// TwinCAT 3 PLC project Untitled1
// ProgramVersion: 3.1.4023.0
// libraries:
//   Tc2_MC2, * (Beckhoff Automation GmbH)
//   Tc2_MC2_Drive, * (Beckhoff Automation GmbH)
//   Tc2_NC, * (Beckhoff Automation GmbH)
//   Tc2_Standard, * (Beckhoff Automation GmbH)
//   Tc2_System, * (Beckhoff Automation GmbH)
//   Tc3_Module, * (Beckhoff Automation GmbH)
// project tree:
//   GVLs/ link.TcGVL (not stored)
//   / PlcTask.TcTTO
//   POUs/ ControlParameters.TcPOU, ImpulseTest.TcPOU, leastSquare.TcPOU, MAIN.TcPOU, TorqueCounnter.TcPOU, torqueInput.TcPOU, velocityInput.TcPOU, velocityInput_.TcPOU, VelocityRide.TcPOU
// real-time tasks:
//   TASK PlcTask: cycle T#1ms, priority 8, ADS port 350
// motion (NC):
//   TASK NC-Task 1 SAF: cycle T#1ms, priority 4, ADS port 501
//   TASK NC-Task 1 SVB: cycle T#10ms, priority 10, ADS port 511
//   AXIS Axis 1 (id 1)
//     Dynamic: Acceleration=417.42, Deceleration=417.42, Jerk=1252.26
//     Velo: RefSearch=2.7828, RefSync=2.7828, SlowManual=13.914, FastManual=83.484, Fast=278.28, Maximum=278.28
//     OtherSettings: AllowMotionCmdToSlave=true
//     encoder EncType=19
//       EncPara: ScaleFactorNumerator=5, ScaleFactorDenominator=1048576, MaxCount=#xffffffff
//     drive DrvType=16
//       DrvPara: MaxCount=#xffffffff, DriveControlDWord=#x00020000
//         Analog: VeloReferenz=306.108, VeloScale=71.5255737304688, TorqueSetpointScale=10, ScaleFactorActTorque=0.1
//         TimeComp: TaskDelayCycles=1
//     controller CtrType=1
//       CtrPara: PriorControlFactor=1
//         PosDiffControl: Enable=false
//         Observer: BandWidth=20
//   AXIS Axis 2 (id 2)
//     Dynamic: Acceleration=417.42, Deceleration=417.42, Jerk=1252.26
//     Velo: RefSearch=2.7828, RefSync=2.7828, SlowManual=13.914, FastManual=83.484, Fast=278.28, Maximum=278.28
//     OtherSettings: AllowMotionCmdToSlave=true
//     encoder EncType=19
//       EncPara: ScaleFactorNumerator=5, ScaleFactorDenominator=1048576, MaxCount=#xffffffff
//     drive DrvType=16
//       DrvPara: MaxCount=#xffffffff, DriveControlDWord=#x00020000
//         Analog: VeloReferenz=306.108, VeloScale=71.5255737304688, TorqueSetpointScale=10, ScaleFactorActTorque=0.1
//         TimeComp: TaskDelayCycles=1
//     controller CtrType=1
//       CtrPara: PriorControlFactor=1
//         PosDiffControl: Enable=false
//         Observer: BandWidth=20
//   AXIS Axis 3 (id 3)
//     Dynamic: Acceleration=417.42, Deceleration=417.42, Jerk=1252.26
//     Velo: RefSearch=2.7828, RefSync=2.7828, SlowManual=13.914, FastManual=83.484, Fast=278.28, Maximum=278.28
//     OtherSettings: AllowMotionCmdToSlave=true
//     encoder EncType=19
//       EncPara: ScaleFactorNumerator=5, ScaleFactorDenominator=1048576, MaxCount=#xffffffff
//     drive DrvType=16
//       DrvPara: MaxCount=#xffffffff, DriveControlDWord=#x00000100
//         Analog: VeloReferenz=306.108, VeloScale=71.5255737304688, TorqueSetpointScale=10, ScaleFactorActTorque=0.1
//         TimeComp: TaskDelayCycles=1
//     controller CtrType=1
//       CtrPara: PriorControlFactor=1
//         Observer: BandWidth=20
//   AXIS Axis 4 (id 4)
//     OtherSettings: AllowMotionCmdToSlave=true
//     encoder EncType=19
//       EncPara: MaxCount=#xffffffff
//     drive DrvType=16
//       DrvPara: MaxCount=#xffffffff, DriveControlDWord=#x00000100
//         Analog: TorqueSetpointScale=10, ScaleFactorActTorque=0.1
//         TimeComp: TaskDelayCycles=1
//     controller CtrType=1
//       CtrPara: PriorControlFactor=1
//         Observer: BandWidth=20
// I/O:
//   DEVICE Device 5 (EtherCAT), AmsNetId 172.18.238.10.6.1
//     Term 1 (EK1100) [EK1100 EtherCAT Coupler (2A E-Bus)]
//       Term 2 (EL9221-5000) [EL9221-5000 Overcurrent protection 24V DC, 1Ch., max. 10A, adjustable]
//       Term 3 (EL1809) [EL1809 16Ch. Dig. Input 24V, 3ms]
//       Term 4 (EL2809) [EL2809 16Ch. Dig. Output 24V, 0.5A]
//       Term 5 (EL4028) [EL4028 8Ch. Ana. Output 4-20mA, 12bit]
//       Term 6 (EL3058) [EL3058 8Ch. Ana. Input 4-20mA]
//       Term 7 (EL3068) [EL3068 8Ch. Ana. Input 0-10V]
//       Term 8 (EL4008) [EL4008 8Ch. Ana. Output 0-10V, 12bit]
//       Term 9 (EL2634) [EL2634 4Ch. Relay Output, NO (250V AC / 30V DC)]
//       Term 10 (EL2634) [EL2634 4Ch. Relay Output, NO (250V AC / 30V DC)]
//       Term 11 (EL2634) [EL2634 4Ch. Relay Output, NO (250V AC / 30V DC)]
//       Term 15 (EL9011) [EL9011 End Terminal]
//     Term 12 (AX8640-0000-0103) [AX8640-0000-0103]
//       Drive 13 (AX8206-0000-0103) [AX8206-0000-0103]
//         modules: Device, Device, Device, Device, Device, Device, Device, Device, Device, Device, Device, Device, Device, Device, Device, Device, Device, Device, Device, Device, Device, Device, Device, Device, Device, Device, Device, Device, Device, Device, Device, Ch A, Ch A, Ch A, Ch A, Ch A, Ch A, Ch A, Ch A, Ch A, Ch A, Ch A, Ch A, Ch A, Ch A, Ch A, Ch A, Ch A, Ch A, Ch A, Ch A, Ch A, Ch A, Ch A, Ch A, Ch A, Ch A, Ch A, Ch B, Ch B, Ch B, Ch B, Ch B, Ch B, Ch B, Ch B, Ch B, Ch B, Ch B, Ch B, Ch B, Ch B, Ch B, Ch B, Ch B, Ch B, Ch B, Ch B, Ch B, Ch B, Ch B, Ch B, Ch B, Ch B, Ch B
//         startup 12992:1 := 414D383034312D78447830 // Ch A Motor parameters / Configured motor type
//         startup 24768:0 := FEFF // Ch A Interpolation sub mode select
//         startup 13000:5 := 0200 // Ch A Motor thermal model / Reaction
//         startup 12992:12 := 00803B45 // Ch A Motor parameters / Motor rated speed
//         startup 12992:13 := BC741340 // Ch A Motor parameters / Motor rated torque
//         startup 24694:0 := 48090000 // Ch A Motor standstill torque
//         startup 24800:0 := D007 // Ch A Positive torque/force limit value
//         startup 24801:0 := D007 // Ch A Negative torque/force limit value
//         startup 12288:6 := 4158383230362D303030302D30303030 // Ch A AxisMain parameters / Configured drive type
//         startup 12867:1 := 3333D33F // Ch A TorqueCtrl parameters / Configured channel rated current
//         startup 12867:2 := 66669E40 // Ch A TorqueCtrl parameters / Configured channel peak current
//         startup 12864:1 := C1059543 // Ch A TorqueCtrl parameters mappable / Torque control proportional gain q
//         startup 12864:2 := 8A0E7C39 // Ch A TorqueCtrl parameters mappable / Torque control integral action time q
//         startup 12608:1 := B246513D // Ch A VeloCtrl parameters mappable / Velocity control proportional gain
//         startup 12608:2 := 6F12033C // Ch A VeloCtrl parameters mappable / Velocity control integral action time
//         startup 12608:3 := 00980546 // Ch A VeloCtrl parameters mappable / Bipolar velocity limit value
//         startup 12992:15 := 0100 // Ch A Motor parameters / Motor temperature sensor connection
//         startup 12611:4 := 0100 // Ch A VeloCtrl observer / Observer type
//         startup 24672:0 := 08 // Ch A Modes of operation
//         startup 12296:2 := 00 // Ch A AxisMain parameters encoder polarity / Primary encoder actual values
//         startup 14016:1 := 414D383034312D78447830 // Ch B Motor parameters / Configured motor type
//         startup 26816:0 := FEFF // Ch B Interpolation sub mode select
//         startup 14024:5 := 0200 // Ch B Motor thermal model / Reaction
//         startup 14016:12 := 00803B45 // Ch B Motor parameters / Motor rated speed
//         startup 14016:13 := BC741340 // Ch B Motor parameters / Motor rated torque
//         startup 26742:0 := 48090000 // Ch B Motor standstill torque
//         startup 26848:0 := D007 // Ch B Positive torque/force limit value
//         startup 26849:0 := D007 // Ch B Negative torque/force limit value
//         startup 13312:6 := 4158383230362D303030302D30303030 // Ch B AxisMain parameters / Configured drive type
//         startup 13891:1 := 3333D33F // Ch B TorqueCtrl parameters / Configured channel rated current
//         startup 13891:2 := 66669E40 // Ch B TorqueCtrl parameters / Configured channel peak current
//         startup 13888:1 := C1059543 // Ch B TorqueCtrl parameters mappable / Torque control proportional gain q
//         startup 13888:2 := 8A0E7C39 // Ch B TorqueCtrl parameters mappable / Torque control integral action time q
//         startup 13632:1 := B246513D // Ch B VeloCtrl parameters mappable / Velocity control proportional gain
//         startup 13632:2 := 6F12033C // Ch B VeloCtrl parameters mappable / Velocity control integral action time
//         startup 13632:3 := 00980546 // Ch B VeloCtrl parameters mappable / Bipolar velocity limit value
//         startup 14016:15 := 0100 // Ch B Motor parameters / Motor temperature sensor connection
//         startup 13635:4 := 0100 // Ch B VeloCtrl observer / Observer type
//         startup 26720:0 := 08 // Ch B Modes of operation
//         startup 13320:2 := 00 // Ch B AxisMain parameters encoder polarity / Primary encoder actual values
//       Drive 14 (AX8206-0000-0103) [AX8206-0000-0103]
//         modules: Device, Device, Device, Device, Device, Device, Device, Device, Device, Device, Device, Device, Device, Device, Device, Device, Device, Device, Device, Device, Device, Device, Device, Device, Device, Device, Device, Device, Device, Device, Device, Ch A, Ch A, Ch A, Ch A, Ch A, Ch A, Ch A, Ch A, Ch A, Ch A, Ch A, Ch A, Ch A, Ch A, Ch A, Ch A, Ch A, Ch A, Ch A, Ch A, Ch A, Ch A, Ch A, Ch A, Ch A, Ch A, Ch A, Ch B, Ch B, Ch B, Ch B, Ch B, Ch B, Ch B, Ch B, Ch B, Ch B, Ch B, Ch B, Ch B, Ch B, Ch B, Ch B, Ch B, Ch B, Ch B, Ch B, Ch B, Ch B, Ch B, Ch B, Ch B, Ch B
//         startup 12992:1 := 414D383034312D78447831 // Ch A Motor parameters / Configured motor type
//         startup 24768:0 := FEFF // Ch A Interpolation sub mode select
//         startup 13000:5 := 0200 // Ch A Motor thermal model / Reaction
//         startup 12992:12 := 00803B45 // Ch A Motor parameters / Motor rated speed
//         startup 12992:13 := BC741340 // Ch A Motor parameters / Motor rated torque
//         startup 24694:0 := 48090000 // Ch A Motor standstill torque
//         startup 24800:0 := D007 // Ch A Positive torque/force limit value
//         startup 24801:0 := D007 // Ch A Negative torque/force limit value
//         startup 12288:6 := 4158383230362D303030302D30303030 // Ch A AxisMain parameters / Configured drive type
//         startup 12867:1 := 3333D33F // Ch A TorqueCtrl parameters / Configured channel rated current
//         startup 12867:2 := 66669E40 // Ch A TorqueCtrl parameters / Configured channel peak current
//         startup 12864:1 := C1059543 // Ch A TorqueCtrl parameters mappable / Torque control proportional gain q
//         startup 12864:2 := 8A0E7C39 // Ch A TorqueCtrl parameters mappable / Torque control integral action time q
//         startup 12608:1 := 7409A73D // Ch A VeloCtrl parameters mappable / Velocity control proportional gain
//         startup 12608:2 := 6F12033C // Ch A VeloCtrl parameters mappable / Velocity control integral action time
//         startup 12608:3 := 00980546 // Ch A VeloCtrl parameters mappable / Bipolar velocity limit value
//         startup 12992:15 := 0100 // Ch A Motor parameters / Motor temperature sensor connection
//         startup 12611:4 := 0100 // Ch A VeloCtrl observer / Observer type
//         startup 24672:0 := 08 // Ch A Modes of operation
//         startup 12296:2 := 00 // Ch A AxisMain parameters encoder polarity / Primary encoder actual values
//       Term 16 (EL9011) [EL9011 End Terminal]
// variable links:
//   Device 5 (EtherCAT) <-> Device 5 (EtherCAT)/Term 12 (AX8640-0000-0103)/Drive 13 (AX8206-0000-0103)
//     Term 12 (AX8640-0000-0103)/PSM Controlword for axis/Controlword for axis <-> Device/DeviceMain Outputs/Power supply controlword
//   Device 5 (EtherCAT) <-> Device 5 (EtherCAT)/Term 12 (AX8640-0000-0103)/Drive 14 (AX8206-0000-0103)
//     Term 12 (AX8640-0000-0103)/PSM Controlword for axis/Controlword for axis <-> Device/DeviceMain Outputs/Power supply controlword
//   NC-Task 1 SAF/Axes/Axis 1 <-> Device 5 (EtherCAT)/Term 12 (AX8640-0000-0103)/Drive 13 (AX8206-0000-0103)
//     Drive/Inputs/In/nDataIn1 <-> Ch A/Ch A PositionControl Inputs/Ch A Following error actual value
//     Drive/Inputs/In/nDataIn3[0] <-> Ch A/Ch A TorqueControl Inputs/Ch A Torque/force actual value
//     Drive/Inputs/In/nDcOutputTime <-> InfoData/DcOutputShift
//     Drive/Inputs/In/nState1 <-> Ch A/Ch A AxisMain Inputs/Ch A Statusword
//     Drive/Inputs/In/nState2 <-> Ch A/Ch A AxisMain Inputs/Ch A Statusword @bit 8
//     Drive/Inputs/In/nState4 @bit 1 <-> WcState/InputToggle
//     Drive/Inputs/In/nState4 <-> WcState/WcState
//     Drive/Outputs/Out/nCtrl1 <-> Ch A/Ch A AxisMain Outputs/Ch A Controlword
//     Drive/Outputs/Out/nCtrl2 <-> Ch A/Ch A AxisMain Outputs/Ch A Controlword @bit 8
//     Drive/Outputs/Out/nDataOut1 <-> Ch A/Ch A Interpolator Outputs/Ch A Target position
//     Enc/Inputs/In/nDataIn1 <-> Ch A/Ch A AxisMain Inputs/Ch A Position actual value
//     Enc/Inputs/In/nDataIn7 <-> Ch A/Ch A AxisMain Inputs/Ch A Velocity actual value
//     Enc/Inputs/In/nDcInputTime <-> InfoData/DcInputShift
//     Enc/Inputs/In/nState2 @bit 5 <-> Ch A/Ch A AxisMain Inputs/Position actual value invalid
//     Enc/Inputs/In/nState4 @bit 1 <-> WcState/InputToggle
//     Enc/Inputs/In/nState4 <-> WcState/WcState
//   NC-Task 1 SAF/Axes/Axis 2 <-> Device 5 (EtherCAT)/Term 12 (AX8640-0000-0103)/Drive 13 (AX8206-0000-0103)
//     Drive/Inputs/In/nDataIn1 <-> Ch B/Ch B PositionControl Inputs/Ch B Following error actual value
//     Drive/Inputs/In/nDataIn3[0] <-> Ch B/Ch B TorqueControl Inputs/Ch B Torque/force actual value
//     Drive/Inputs/In/nDcOutputTime <-> InfoData/DcOutputShift
//     Drive/Inputs/In/nState1 <-> Ch B/Ch B AxisMain Inputs/Ch B Statusword
//     Drive/Inputs/In/nState2 <-> Ch B/Ch B AxisMain Inputs/Ch B Statusword @bit 8
//     Drive/Inputs/In/nState4 @bit 1 <-> WcState/InputToggle
//     Drive/Inputs/In/nState4 <-> WcState/WcState
//     Drive/Outputs/Out/nCtrl1 <-> Ch B/Ch B AxisMain Outputs/Ch B Controlword
//     Drive/Outputs/Out/nCtrl2 <-> Ch B/Ch B AxisMain Outputs/Ch B Controlword @bit 8
//     Drive/Outputs/Out/nDataOut1 <-> Ch B/Ch B Interpolator Outputs/Ch B Target position
//     Enc/Inputs/In/nDataIn1 <-> Ch B/Ch B AxisMain Inputs/Ch B Position actual value
//     Enc/Inputs/In/nDataIn7 <-> Ch B/Ch B AxisMain Inputs/Ch B Velocity actual value
//     Enc/Inputs/In/nDcInputTime <-> InfoData/DcInputShift
//     Enc/Inputs/In/nState2 @bit 5 <-> Ch B/Ch B AxisMain Inputs/Position actual value invalid
//     Enc/Inputs/In/nState4 @bit 1 <-> WcState/InputToggle
//     Enc/Inputs/In/nState4 <-> WcState/WcState
//   NC-Task 1 SAF/Axes/Axis 3 <-> Device 5 (EtherCAT)/Term 12 (AX8640-0000-0103)/Drive 14 (AX8206-0000-0103)
//     Drive/Inputs/In/nDataIn1 <-> Ch A/Ch A PositionControl Inputs/Ch A Following error actual value
//     Drive/Inputs/In/nDataIn3[0] <-> Ch A/Ch A TorqueControl Inputs/Ch A Torque/force actual value
//     Drive/Inputs/In/nDcOutputTime <-> InfoData/DcOutputShift
//     Drive/Inputs/In/nState1 <-> Ch A/Ch A AxisMain Inputs/Ch A Statusword
//     Drive/Inputs/In/nState2 <-> Ch A/Ch A AxisMain Inputs/Ch A Statusword @bit 8
//     Drive/Inputs/In/nState4 @bit 1 <-> WcState/InputToggle
//     Drive/Inputs/In/nState4 <-> WcState/WcState
//     Drive/Outputs/Out/nCtrl1 <-> Ch A/Ch A AxisMain Outputs/Ch A Controlword
//     Drive/Outputs/Out/nCtrl2 <-> Ch A/Ch A AxisMain Outputs/Ch A Controlword @bit 8
//     Enc/Inputs/In/nDataIn1 <-> Ch A/Ch A AxisMain Inputs/Ch A Position actual value
//     Enc/Inputs/In/nDataIn7 <-> Ch A/Ch A AxisMain Inputs/Ch A Velocity actual value
//     Enc/Inputs/In/nDcInputTime <-> InfoData/DcInputShift
//     Enc/Inputs/In/nState2 @bit 5 <-> Ch A/Ch A AxisMain Inputs/Position actual value invalid
//     Enc/Inputs/In/nState4 @bit 1 <-> WcState/InputToggle
//     Enc/Inputs/In/nState4 <-> WcState/WcState
//   NC-Task 1 SAF/Axes/Axis 4 <-> Device 5 (EtherCAT)/Term 12 (AX8640-0000-0103)/Drive 14 (AX8206-0000-0103)
//     Drive/Inputs/In/nDataIn1 <-> Ch B/Ch B PositionControl Inputs/Ch B Following error actual value
//     Drive/Inputs/In/nState1 <-> Ch B/Ch B AxisMain Inputs/Ch B Statusword
//     Drive/Inputs/In/nState2 <-> Ch B/Ch B AxisMain Inputs/Ch B Statusword @bit 8
//     Drive/Outputs/Out/nCtrl1 <-> Ch B/Ch B AxisMain Outputs/Ch B Controlword
//     Drive/Outputs/Out/nCtrl2 <-> Ch B/Ch B AxisMain Outputs/Ch B Controlword @bit 8
//     Enc/Inputs/In/nDataIn1 <-> Ch B/Ch B AxisMain Inputs/Ch B Position actual value
//     Enc/Inputs/In/nState2 @bit 5 <-> Ch B/Ch B AxisMain Inputs/Position actual value invalid
//   Untitled1/Untitled1 Instance <-> Device 5 (EtherCAT)/Term 12 (AX8640-0000-0103)/Drive 13 (AX8206-0000-0103)
//     PlcTask Outputs/link.torqueOfsetX <-> Ch A/Ch A TorqueControl Outputs/Ch A Torque/force offset
//     PlcTask Outputs/link.torqueOfsetY <-> Ch B/Ch B TorqueControl Outputs/Ch B Torque/force offset
//     PlcTask Outputs/link.torqueX <-> Ch A/Ch A TorqueControl Outputs/Ch A Target torque/force
//     PlcTask Outputs/link.torqueY <-> Ch B/Ch B TorqueControl Outputs/Ch B Target torque/force
//     PlcTask Outputs/link.xAxisVelocity <-> Ch A/Ch A Interpolator Outputs/Ch A Target velocity
//     PlcTask Outputs/link.yAxisVelocity <-> Ch B/Ch B Interpolator Outputs/Ch B Target velocity
//   Untitled1/Untitled1 Instance <-> Device 5 (EtherCAT)/Term 12 (AX8640-0000-0103)/Drive 14 (AX8206-0000-0103)
//     PlcTask Outputs/link.zAxisVelocity <-> Ch A/Ch A Interpolator Outputs/Ch A Target velocity
//   Untitled1/Untitled1 Instance <-> NC-Task 1 SAF/Axes/Axis 1
//     PlcTask Inputs/MAIN.setAxis[0].NcToPlc <-> Outputs/ToPlc
//     PlcTask Outputs/MAIN.setAxis[0].PlcToNc <-> Inputs/FromPlc
//   Untitled1/Untitled1 Instance <-> NC-Task 1 SAF/Axes/Axis 2
//     PlcTask Inputs/MAIN.setAxis[1].NcToPlc <-> Outputs/ToPlc
//     PlcTask Outputs/MAIN.setAxis[1].PlcToNc <-> Inputs/FromPlc
//   Untitled1/Untitled1 Instance <-> NC-Task 1 SAF/Axes/Axis 3
//     PlcTask Inputs/MAIN.setAxis[2].NcToPlc <-> Outputs/ToPlc
//     PlcTask Outputs/MAIN.setAxis[2].PlcToNc <-> Inputs/FromPlc

CONFIGURATION Untitled1
    RESOURCE PLC ON TwinCAT3
        TASK PlcTask(INTERVAL := T#500us, PRIORITY := 8);
        PROGRAM MAIN WITH PlcTask : MAIN;
        PROGRAM leastSquare WITH PlcTask : leastSquare;
        PROGRAM velocityInput_ WITH PlcTask : velocityInput_;
        PROGRAM velocityInput WITH PlcTask : velocityInput;
        PROGRAM torqueInput WITH PlcTask : torqueInput;
        PROGRAM ImpulseTest WITH PlcTask : ImpulseTest;
        PROGRAM VelocityRide WITH PlcTask : VelocityRide;
    END_RESOURCE
END_CONFIGURATION

// ---- POUs/MAIN.TcPOU
PROGRAM MAIN
VAR
	sampleTime: REAL := 0.5;
	state: INT	:=	0;	
	start: BOOL	:=	FALSE;
	operationModeWrite: SINT	:=	10;	
	
	{attribute 'TcNcAxis' := '[0]:=Axis 1;[1]:=Axis 2;[2]:=Axis 3'} 
    // Using an axis in an array.
    setAxis     : ARRAY [0..2] OF AXIS_REF;
	
	opertionModeRead: SINT;
	
	fbCoERead: FB_CoERead;
	
	MotorEnable: BOOL:=FALSE;
	
	mcReset: MC_Reset;
	mcPower: MC_Power;
	
////////
	
	operitonModeCh: WORD;
	subIndex: BYTE;	
	axisSelect: (xAxis, yAxis, zAxis, xyAxis, allAxis);	
	fbCoEWrite: FB_CoEWrite;	
	//torque : FB_TorqueInput;
	
END_VAR
VAR_INPUT
	dummy : INT ;
END_VAR

CASE state OF
	//Axis Selection
0:
	IF start THEN
		
		IF axisSelect = xAxis THEN
			operitonModeCh := 16#6060;
			subIndex := 0;
			MotorEnable:=TRUE;
			dummy := 0;	
		ELSIF axisSelect = yAxis THEN	
			operitonModeCh := 16#6860;		
			subIndex := 0;
			MotorEnable:=TRUE;	
			dummy := 1;	
		ELSIF axisSelect = zAxis THEN	
			operitonModeCh := 16#6860;
			MotorEnable:=TRUE;	
			dummy := 2;
			subIndex := 0;
			
		ELSIF axisSelect = xyAxis THEN	
			operitonModeCh := 16#6860;
			MotorEnable:=TRUE;	
			dummy := 3;
			subIndex := 0;
		END_IF
		
		state:=190;
		start:=FALSE;		
	END_IF

190:
	mcReset(
	Axis:=setAxis[dummy] , 
	Execute:=TRUE , 
	 );
	IF NOT mcReset.Busy AND mcReset.Done THEN		
		mcReset(Axis:=setAxis[dummy], Execute:=FALSE);		
		state:=200;
	END_IF
	
	//Mod of operation
200:


	fbCoEWrite(
		Axis:= setAxis[dummy], 
		NetId:='', 
		Index:= operitonModeCh, 
		SubIndex:=subIndex,
		pSrcBuf:= ADR(operationModeWrite), 
		BufLen:= SIZEOF(operationModeWrite), 
		Execute:=TRUE , 		
		CompleteAccess:=TRUE , 
		 );
		
	IF NOT fbCoEWrite.Busy THEN
		fbCoEWrite(
		Axis:= setAxis[dummy], 
		NetId:='', 
		Index:= operitonModeCh, 
		SubIndex:=subIndex, 
		pSrcBuf:= ADR(operationModeWrite), 
		BufLen:= SIZEOF(operationModeWrite), 
		Execute:=FALSE , 		
		CompleteAccess:=TRUE , 
		 );
		
		fbCoERead(
			Axis:=setAxis[dummy] , 
			NetId:= '', 
			Index:= operitonModeCh,
			SubIndex:= subIndex,
			pDstBuf:= ADR(opertionModeRead), 
			BufLen:= SIZEOF(opertionModeRead), 
			Execute:= TRUE, 			
			CompleteAccess:=TRUE , 
			 );
			
			IF opertionModeRead = operationModeWrite AND NOT fbCoERead.Busy THEN
			
				fbCoeRead(Axis:=setAxis[dummy],Execute:=FALSE );
				IF NOT fbCoERead.Execute THEN
					state:=210;
				END_IF
			END_IF
	END_IF
	
	//power enable
	//motor enable
210:
	mcReset(
	Axis:=setAxis[dummy] , 
	Execute:=TRUE , 
	 );
	IF NOT mcReset.Busy AND mcReset.Done THEN		
		mcReset(Axis:=setAxis[dummy], Execute:=FALSE);		
		state:=220;
	END_IF
	
	220:
	
	mcPower(
	Axis:=setAxis[dummy] , 
	Enable:= MotorEnable , 
	Enable_Positive:= MotorEnable, 
	Enable_Negative:= MotorEnable, 
 );
	IF (mcPower.Status AND MotorEnable) OR (NOT mcPower.Status AND NOT MotorEnable) THEN 

		state:=230;
	END_IF
	

230:

// 	torque(torqueInput:=20, duration:=2);
//	IF torque.busy = FALSE THEN
//		state := 232;
//	END_IF

 
232:
  
// velocityInput();
// IF NOT velocityInput.busy THEN
//	 state := 240;
// END_IF
 
240 :
 mcReset(
	Axis:=setAxis[dummy] , 
	Execute:=TRUE , 
	 );
	IF NOT mcReset.Busy AND mcReset.Done THEN		
		mcReset(Axis:=setAxis[dummy], Execute:=FALSE);		
		state:=250;
	END_IF
 
	250:
 	MotorEnable := FALSE;
 	mcPower(
	Axis:=setAxis[dummy] , 
	Enable:= MotorEnable , 
	Enable_Positive:= MotorEnable, 
	Enable_Negative:= MotorEnable, 
 );
	IF (mcPower.Status AND MotorEnable) OR (NOT mcPower.Status AND NOT MotorEnable) THEN 
		state:=260;
	END_IF
	//Motor disable
260:
 	

	state := 0;

END_CASE

END_PROGRAM

// ---- POUs/leastSquare.TcPOU
PROGRAM leastSquare
VAR
	state: USINT := 0;
	Torque_Nm :REAL := 0.5;
	duration :INT :=10000;
	startTest :BOOL := FALSE;	
	TorquePerThousand: INT;		

	TorqueCounter: INT;
	TorqInterval: INT;
END_VAR

CASE state OF
	
0 :
	
	IF MAIN.dummy = 0 AND startTest  THEN
		state := 10;
	ELSIF MAIN.dummy = 1 AND startTest THEN
		state := 30;
	END_IF	

	10: //varying amplitude squarewaves for least square
			IF startTest THEN
				TorqueCounter := TorqueCounter + 1;
				IF TorqueCounter < TorqInterval THEN
					link.torqueX := TO_INT(Torque_Nm * 1/2.37*1000);
				ELSIF TorqueCounter >= TorqInterval AND TorqueCounter <TorqInterval*2 THEN
					link.torqueX := TO_INT(-Torque_Nm *1/2.37*1000);
				ELSIF TorqueCounter >= TorqInterval*2 AND TorqueCounter <TorqInterval*3 THEN
					link.torqueX := TO_INT(Torque_Nm * 2/2.37*1000); 
				ELSIF TorqueCounter >= TorqInterval*3 AND TorqueCounter <TorqInterval*4 THEN
					link.torqueX := TO_INT(-Torque_Nm * 2/2.37*1000);
				ELSIF TorqueCounter >= TorqInterval*4 AND TorqueCounter <TorqInterval*5 THEN
					link.torqueX := TO_INT(Torque_Nm * 3/2.37*1000); 
				ELSIF TorqueCounter >= TorqInterval*5 AND TorqueCounter <TorqInterval*6 THEN
					link.torqueX := TO_INT(-Torque_Nm * 3/2.37*1000);
				ELSIF TorqueCounter >= TorqInterval*6 AND TorqueCounter <TorqInterval*7 THEN
					link.torqueX := TO_INT(Torque_Nm * 4/2.37*1000); 
					
				ELSIF TorqueCounter >= TorqInterval*7 AND TorqueCounter <TorqInterval*8 THEN
					link.torqueX := TO_INT(-Torque_Nm * 4/2.37*1000);		
				ELSIF TorqueCounter >= TorqInterval*8 AND TorqueCounter <TorqInterval*9 THEN
					link.torqueX := TO_INT(Torque_Nm * 3/2.37*1000); 
				ELSIF TorqueCounter >= TorqInterval*9 AND TorqueCounter <TorqInterval*10 THEN
					link.torqueX := TO_INT(-Torque_Nm * 3/2.37*1000);
				ELSIF TorqueCounter >= TorqInterval*10 AND TorqueCounter <TorqInterval*11 THEN
					link.torqueX := TO_INT(Torque_Nm * 2/2.37*1000); 
				ELSIF TorqueCounter >= TorqInterval*11 AND TorqueCounter <TorqInterval*12 THEN
					link.torqueX := TO_INT(-Torque_Nm * 2/2.37*1000);
				ELSIF TorqueCounter >= TorqInterval*12 AND TorqueCounter <TorqInterval*13 THEN
					link.torqueX := TO_INT(Torque_Nm * 1/2.37*1000); 
				ELSIF TorqueCounter >= TorqInterval*13 AND TorqueCounter <TorqInterval*14 THEN
					link.torqueX := TO_INT(-Torque_Nm * 1/2.37*1000);
				ELSIF TorqueCounter >= TorqInterval*14 THEN
					link.torqueX := 0;
					state:=60;
				END_IF
		ELSE
		link.torqueX := 0;		
		startTest := FALSE;
		TorqueCounter := 0;
		state := 60;
		
		END_IF
	30: //varying amplitude squarewaves for least square
			IF startTest THEN
				TorqueCounter := TorqueCounter + 1;
				IF TorqueCounter < TorqInterval THEN
					link.torqueY := TO_INT(Torque_Nm * 0.5/2.37*1000);
				ELSIF TorqueCounter >= TorqInterval AND TorqueCounter <TorqInterval*2 THEN
					link.torqueY := TO_INT(-Torque_Nm *0.5/2.37*1000);
				ELSIF TorqueCounter >= TorqInterval*2 AND TorqueCounter <TorqInterval*3 THEN
					link.torqueY := TO_INT(Torque_Nm * 1/2.37*1000); 
				ELSIF TorqueCounter >= TorqInterval*3 AND TorqueCounter <TorqInterval*4 THEN
					link.torqueY := TO_INT(-Torque_Nm * 1/2.37*1000);
				ELSIF TorqueCounter >= TorqInterval*4 AND TorqueCounter <TorqInterval*5 THEN
					link.torqueY := TO_INT(Torque_Nm * 1.5/2.37*1000); 
				ELSIF TorqueCounter >= TorqInterval*5 AND TorqueCounter <TorqInterval*6 THEN
					link.torqueY := TO_INT(-Torque_Nm * 1.5/2.37*1000);
				ELSIF TorqueCounter >= TorqInterval*6 AND TorqueCounter <TorqInterval*7 THEN
					link.torqueY := TO_INT(Torque_Nm * 2/2.37*1000); 
				ELSIF TorqueCounter >= TorqInterval*7 AND TorqueCounter <TorqInterval*8 THEN
					link.torqueY := TO_INT(-Torque_Nm * 2/2.37*1000); 	
				ELSIF TorqueCounter >= TorqInterval*8 AND TorqueCounter <TorqInterval*9 THEN
					link.torqueY := TO_INT(Torque_Nm * 2.5/2.37*1000); 				
				ELSIF TorqueCounter >= TorqInterval*9 AND TorqueCounter <TorqInterval*10 THEN
					link.torqueY := TO_INT(-Torque_Nm * 2.5/2.37*1000); 					

				ELSIF TorqueCounter >= TorqInterval*10 AND TorqueCounter <TorqInterval*11 THEN
					link.torqueY := TO_INT(Torque_Nm * 2/2.37*1000); 					
				ELSIF TorqueCounter >= TorqInterval*11 AND TorqueCounter <TorqInterval*12 THEN
					link.torqueY := TO_INT(-Torque_Nm * 2/2.37*1000);							
				ELSIF TorqueCounter >= TorqInterval*12 AND TorqueCounter <TorqInterval*13 THEN
					link.torqueY := TO_INT(Torque_Nm * 1.5/2.37*1000);			
				ELSIF TorqueCounter >= TorqInterval*13 AND TorqueCounter <TorqInterval*14 THEN
					link.torqueY := TO_INT(-Torque_Nm * 1.5/2.37*1000);		
				ELSIF TorqueCounter >= TorqInterval*14 AND TorqueCounter <TorqInterval*15 THEN
					link.torqueY := TO_INT(Torque_Nm * 1/2.37*1000); 
				ELSIF TorqueCounter >= TorqInterval*15 AND TorqueCounter <TorqInterval*16 THEN
					link.torqueY := TO_INT(-Torque_Nm * 1/2.37*1000);
				ELSIF TorqueCounter >= TorqInterval*16 AND TorqueCounter <TorqInterval*17 THEN
					link.torqueY := TO_INT(Torque_Nm * 0.5/2.37*1000); 
				ELSIF TorqueCounter >= TorqInterval*17 AND TorqueCounter <TorqInterval*18 THEN
					link.torqueY := TO_INT(-Torque_Nm * 0.5/2.37*1000);
				ELSIF TorqueCounter >= TorqInterval*18 THEN
					link.torqueY := 0;
					state:=60;
				END_IF
		ELSE
		link.torqueY := 0;		
		startTest := FALSE;
		TorqueCounter := 0;
		state := 60;
		
		END_IF
	
	
60 :
	startTest:= FALSE;
	state :=0;
	TorqueCounter := 0;
END_CASE

END_PROGRAM

// ---- POUs/velocityInput_.TcPOU
PROGRAM velocityInput_
VAR
	
	velocityStarter : BOOL := FALSE;
	state : INT := 0;	
	counter : LREAL := 0;
	bias : LREAL :=0.4;
	duration: REAL := 30000;
	velocityInput: INT:= -1;
	f0 :LREAL	:=0;
	f1 :LREAL:=100;
	T : LREAL ;	
	x: LREAL;	
	


END_VAR

CASE state OF

0 :
	
	IF MAIN.dummy = 0 AND velocityStarter  THEN
		state := 10;
	ELSIF MAIN.dummy = 1 AND velocityStarter THEN
		state := 30;
	END_IF	
		
10 : 

	IF velocityStarter THEN		
		
		IF counter < duration THEN
			T :=duration/1000.0;
			x:=SIN(2*pi*((f0*counter/1000)+((f1-f0)/(2*T)*(EXPT(counter/1000,2)))));
			link.xAxisVelocity := LREAL_TO_DINT((velocityInput*10000/(5)*60)*(x+bias/(velocityInput)));
		ELSE
			link.xAxisVelocity := 0;
			state := 60;
		END_IF
		counter := counter + MAIN.sampleTime;
	ELSE
		link.xAxisVelocity := 0;
	
	END_IF
	
30:
	IF velocityStarter THEN		
		
		IF counter < duration THEN
			T :=duration/1000.0;
			x:=SIN(2*pi*((f0*counter/1000)+((f1-f0)/(2*T)*(EXPT(counter/1000,2)))));
			link.yAxisVelocity := LREAL_TO_DINT((velocityInput*10000/(5)*60)*(x+bias/(velocityInput)));
		ELSE
			link.yAxisVelocity := 0;
			state := 60;
		END_IF
		counter := counter + MAIN.sampleTime;
	ELSE
		link.yAxisVelocity := 0;
	
	END_IF

60 :
	velocityStarter:= FALSE;
	state :=0;
	counter := 0;
END_CASE

END_PROGRAM

// ---- POUs/velocityInput.TcPOU
PROGRAM velocityInput
VAR
	velocityStarter : BOOL := FALSE;
	state : INT := 0;	
	counter : LREAL := 0;
	
	duration: DINT := 30000;
	velocityInput: INT:= -1;
	
END_VAR

CASE state OF

0 :
	
	IF MAIN.dummy = 0 AND velocityStarter  THEN
		state := 10;
	ELSIF MAIN.dummy = 1 AND velocityStarter THEN
		state := 30;
	END_IF	
		
10 : 

	IF velocityStarter THEN		
		
		IF counter < duration THEN
			link.xAxisVelocity := REAL_TO_DINT(velocityInput*10000/(5)*60);
		ELSE
			link.xAxisVelocity := 0;
			state := 60;
		END_IF
		counter := counter + MAIN.sampleTime;
	ELSE
		link.xAxisVelocity := 0;
	
	END_IF
	
30:
	IF velocityStarter THEN		
		
		IF counter < duration THEN
			link.yAxisVelocity := REAL_TO_DINT(velocityInput*10000/(5)*60);
		ELSE
			link.yAxisVelocity := 0;
			state := 60;
		END_IF
		counter := counter + MAIN.sampleTime;
	ELSE
		link.yAxisVelocity := 0;
	
	END_IF

60 :
	velocityStarter:= FALSE;
	state :=0;
	counter := 0;
END_CASE

END_PROGRAM

// ---- POUs/torqueInput.TcPOU
PROGRAM torqueInput
VAR
	frequency : LREAL :=0 ;
	bias : LREAL :=0.4;
	duration: LREAL := 1000;
	torqueInput: REAL:= 0.05;
	torqueStarter : BOOL:= FALSE;
	state : INT := 10;	
	counter : LREAL := 0;
	f0 :LREAL	:=0;
	f1 :LREAL:=100;
	T : LREAL ;	
	x: LREAL;	
	
END_VAR

CASE state OF
	
10 :
	
	IF MAIN.dummy = 0 AND torqueStarter THEN
		state := 20;
	ELSIF MAIN.dummy = 1 AND torqueStarter THEN
		state := 30;
	END_IF
 
	
20 :
IF 	torqueStarter THEN
	counter := counter + MAIN.sampleTime;
	IF counter < duration THEN
		T :=duration/1000.0;
		frequency := f0 + counter/1000 *(f1-f0)/T;	
		//link.torqueOfsetX := REAL_TO_INT(torqueInput*(1000/2.37));
		x:=SIN(2*pi*((f0*counter/1000)+((f1-f0)/(2*T)*(EXPT(counter/1000,2)))));
			IF MAIN.opertionModeRead=10 THEN
		//link.torqueOfsetX := LREAL_TO_INT(torqueInput*(1000/2.37)*x);
			link.torqueX := LREAL_TO_INT((torqueInput*1000/2.37)*(x+bias/(torqueInput)));
			
			ELSIF MAIN.opertionModeRead=9 THEN				
			link.torqueOfsetX := LREAL_TO_INT(torqueInput*(1000/2.37)*x);
			END_IF
	ELSE
		link.torqueX := 0;
		link.torqueOfsetX := 0;
		torqueStarter := FALSE;
		counter := 0;
		state := 60;
		
	END_IF
ELSE
	link.torqueOfsetX := 0;
END_IF
	
30 :
IF 	torqueStarter THEN
	counter := counter +  MAIN.sampleTime;
	IF counter < duration THEN
		T :=duration/1000.0;
		frequency := f0 + counter/1000.0 *(f1-f0)/T;	
		//link.torqueOfsetY := REAL_TO_INT(torqueInput*(1000/2.37));
		x:=SIN(2*pi*((f0*counter/1000)+((f1-f0)/(2*T)*(EXPT(counter/1000,2)))));
			IF MAIN.opertionModeRead=10 THEN
		//link.torqueOfsetY := LREAL_TO_INT(torqueInput*(1000/2.37)*x);
			link.torqueY := LREAL_TO_INT((torqueInput*1000/2.37)*(x+bias/(torqueInput)));
			
			ELSIF MAIN.opertionModeRead=9 THEN				
			link.torqueOfsetY := LREAL_TO_INT(torqueInput*(1000/2.37)*x);
			END_IF
	ELSE
		link.torqueY := 0;
		link.torqueOfsetY := 0;
		torqueStarter := FALSE;
		counter := 0;
		state := 60;
		
	END_IF
ELSE
	link.torqueOfsetY := 0;
END_IF
60 :
	torqueStarter:=FALSE;
	state :=10;
	counter := 0;
			
	
END_CASE

END_PROGRAM

// ---- POUs/ImpulseTest.TcPOU
PROGRAM ImpulseTest
VAR
	duration: LREAL := 2;
	torqueInput: REAL:= 0.05;
	torqueStarter : BOOL:= FALSE;
	state : INT := 10;	
	counter : LREAL := 0;	
	trial: INT := 5;
	delaytime: LREAL := 5000;
	counter1: LREAL := 0;
	counter3: LREAL :=0;
END_VAR

CASE state OF
10 :

	IF MAIN.dummy = 0 AND torqueStarter THEN
		state := 20;
	ELSIF MAIN.dummy = 1 AND torqueStarter THEN
		state := 30;
	END_IF
	
20 :
IF 	torqueStarter THEN
	counter := counter + MAIN.sampleTime;
	IF counter < duration THEN
			IF MAIN.opertionModeRead=10 THEN
				link.torqueX := REAL_TO_INT(torqueInput*(1000/2.37));	
			ELSIF MAIN.opertionModeRead=9 THEN				
				link.torqueOfsetX := LREAL_TO_INT(torqueInput*(1000/2.37));
			END_IF
	ELSE
		link.torqueX := 0;
		link.torqueOfsetX := 0;
		torqueStarter := FALSE;
		counter := 0;
		counter1:=0;			
		state := 60;
		
	END_IF
ELSE
	link.torqueX := 0;
	link.torqueOfsetX := 0;
END_IF
	
30 :
IF 	torqueStarter THEN
	counter := counter + MAIN.sampleTime;
	IF counter < duration THEN
			IF MAIN.opertionModeRead=10 THEN
				link.torqueY := REAL_TO_INT(torqueInput*(1000/2.37));	
			ELSIF MAIN.opertionModeRead=9 THEN				
				link.torqueOfsetY := LREAL_TO_INT(torqueInput*(1000/2.37));
			END_IF
	ELSE
		link.torqueY := 0;
		link.torqueOfsetY := 0;
		torqueStarter := FALSE;
		counter := 0;
		counter1:=0;		
		state := 60;
		
	END_IF
ELSE
	link.torqueY := 0;
	link.torqueOfsetY := 0;
END_IF

60 :
	counter1:=counter1+  MAIN.sampleTime;
	IF counter1<delaytime THEN
		torqueStarter:=FALSE;	
		counter := 0;
		
		ELSE
			counter3:=counter3+  1;	
			IF counter3 < trial THEN
				torqueStarter:=TRUE;		
				state :=10;
				counter := 0;
			ELSE
				torqueStarter:=FALSE;
				counter3 := 0;		
				state :=10;
				counter := 0;
				counter1 := 0;
				counter3 := 0;
		END_IF
	END_IF
END_CASE

END_PROGRAM

// ---- POUs/VelocityRide.TcPOU
PROGRAM VelocityRide
VAR
	startVelocity: BOOL := FALSE;
	VelocityCounter: DINT;
	VelocityInterval: DINT := 2000;
	VelocityMmPerSecond: DINT := 5;
	
	state: INT := 0;
	
END_VAR

CASE state OF


0 :
	
	IF MAIN.dummy = 0 AND startVelocity  THEN
		state := 10;
	ELSIF MAIN.dummy = 1 AND startVelocity THEN
		state := 30;
	END_IF	
		
10 : 
			IF startVelocity THEN
				VelocityCounter := VelocityCounter + 1;
				IF VelocityCounter < VelocityInterval THEN
					link.xAxisVelocity := TO_DINT((VelocityMmPerSecond + 10 * 0) / 5 * 10000 * 60 );
					
				ELSIF VelocityCounter >= VelocityInterval AND VelocityCounter < VelocityInterval * 2 THEN
					link.xAxisVelocity := TO_DINT(-(VelocityMmPerSecond + 10 * 0) / 5 * 10000 * 60 );
					
				ELSIF VelocityCounter >= VelocityInterval*2 AND VelocityCounter < VelocityInterval*3 THEN
					link.xAxisVelocity := TO_DINT((VelocityMmPerSecond + 10 * 1) / 5 * 10000 * 60 );
 
				ELSIF VelocityCounter >= VelocityInterval*3 AND VelocityCounter < VelocityInterval*4 THEN
					link.xAxisVelocity := TO_DINT(-(VelocityMmPerSecond + 10 * 1) / 5 * 10000 * 60);
					
				ELSIF VelocityCounter >= VelocityInterval*4 AND VelocityCounter < VelocityInterval*5 THEN
					link.xAxisVelocity := TO_DINT((VelocityMmPerSecond + 10 * 2) / 5 * 10000 * 60 );
 
				ELSIF VelocityCounter >= VelocityInterval*5 AND VelocityCounter < VelocityInterval*6 THEN
					link.xAxisVelocity := TO_DINT(-(VelocityMmPerSecond + 10 * 2) / 5 * 10000 * 60);
					
				ELSIF VelocityCounter >= VelocityInterval*6 AND VelocityCounter < VelocityInterval*7 THEN
					link.xAxisVelocity := TO_DINT((VelocityMmPerSecond + 10 * 3) / 5 * 10000 * 60);
					
				ELSIF VelocityCounter >= VelocityInterval*7 AND VelocityCounter < VelocityInterval*8 THEN
					link.xAxisVelocity := TO_DINT(-(VelocityMmPerSecond + 10 * 3) / 5 * 10000 * 60);
					
				ELSIF VelocityCounter >= VelocityInterval*8 AND VelocityCounter < VelocityInterval*9 THEN
					link.xAxisVelocity := TO_DINT((VelocityMmPerSecond + 10 * 4) / 5 * 10000 * 60);
					
				ELSIF VelocityCounter >= VelocityInterval*9 AND VelocityCounter < VelocityInterval*10 THEN
					link.xAxisVelocity := TO_DINT(-(VelocityMmPerSecond + 10 * 4) / 5 * 10000 * 60);
					
				ELSIF VelocityCounter >= VelocityInterval*10 AND VelocityCounter < VelocityInterval*11 THEN
					link.xAxisVelocity := TO_DINT((VelocityMmPerSecond + 10 * 5) / 5 * 10000 * 60);
					
				ELSIF VelocityCounter >= VelocityInterval*11 AND VelocityCounter < VelocityInterval*12 THEN
					link.xAxisVelocity := TO_DINT(-(VelocityMmPerSecond + 10 * 5) / 5 * 10000 * 60);
					
				ELSIF VelocityCounter >= VelocityInterval*12 AND VelocityCounter < VelocityInterval*13 THEN
					link.xAxisVelocity := TO_DINT((VelocityMmPerSecond + 10 * 6) / 5 * 10000 * 60);
					
				ELSIF VelocityCounter >= VelocityInterval*13 AND VelocityCounter < VelocityInterval*14 THEN
					link.xAxisVelocity := TO_DINT(-(VelocityMmPerSecond + 10 * 6) / 5 * 10000 * 60);
					
				ELSIF VelocityCounter >= VelocityInterval*14 AND VelocityCounter < VelocityInterval*15 THEN
					link.xAxisVelocity := TO_DINT((VelocityMmPerSecond + 10 * 7) / 5 * 10000 * 60);
					
				ELSIF VelocityCounter >= VelocityInterval*15 AND VelocityCounter < VelocityInterval*16 THEN
					link.xAxisVelocity := TO_DINT(-(VelocityMmPerSecond + 10 * 7) / 5 * 10000 * 60);
					
				ELSIF VelocityCounter >= VelocityInterval*16 AND VelocityCounter < VelocityInterval*17 THEN
					link.xAxisVelocity := TO_DINT((VelocityMmPerSecond + 10 * 8) / 5 * 10000 * 60);
					
				ELSIF VelocityCounter >= VelocityInterval*17 AND VelocityCounter < VelocityInterval*18 THEN
					link.xAxisVelocity := TO_DINT(-(VelocityMmPerSecond + 10 * 8) / 5 * 10000 * 60);
					
				ELSIF VelocityCounter >= VelocityInterval*18 AND VelocityCounter < VelocityInterval*19 THEN
					link.xAxisVelocity := TO_DINT((VelocityMmPerSecond + 10 * 9) / 5 * 10000 * 60);
					
				ELSIF VelocityCounter >= VelocityInterval*19 AND VelocityCounter < VelocityInterval*20 THEN
					link.xAxisVelocity := TO_DINT(-(VelocityMmPerSecond + 10 * 9) / 5 * 10000 * 60);
					
				ELSIF VelocityCounter >= VelocityInterval*20 AND VelocityCounter < VelocityInterval*21 THEN
					link.xAxisVelocity := TO_DINT((VelocityMmPerSecond + 10 * 10) / 5 * 10000 * 60);
					
				ELSIF VelocityCounter >= VelocityInterval*21 AND VelocityCounter < VelocityInterval*22 THEN
					link.xAxisVelocity := TO_DINT(-(VelocityMmPerSecond + 10 * 10) / 5 * 10000 * 60);
					
				ELSIF VelocityCounter >= VelocityInterval*22 THEN
					link.xAxisVelocity := 0;
					startVelocity := 0;
					state := 60;
					
				END_IF
			ELSE
				state := 60;
			END_IF
			
30 : 
			IF startVelocity THEN
				VelocityCounter := VelocityCounter + 1;
				IF VelocityCounter < VelocityInterval THEN
					link.yAxisVelocity := TO_DINT((VelocityMmPerSecond + 10 * 0) / 5 * 10000 * 60 );
					
				ELSIF VelocityCounter >= VelocityInterval AND VelocityCounter < VelocityInterval * 2 THEN
					link.yAxisVelocity := TO_DINT(-(VelocityMmPerSecond + 10 * 0) / 5 * 10000 * 60 );
					
				ELSIF VelocityCounter >= VelocityInterval*2 AND VelocityCounter < VelocityInterval*3 THEN
					link.yAxisVelocity := TO_DINT((VelocityMmPerSecond + 10 * 1) / 5 * 10000 * 60 );
 
				ELSIF VelocityCounter >= VelocityInterval*3 AND VelocityCounter < VelocityInterval*4 THEN
					link.yAxisVelocity := TO_DINT(-(VelocityMmPerSecond + 10 * 1) / 5 * 10000 * 60);
					
				ELSIF VelocityCounter >= VelocityInterval*4 AND VelocityCounter < VelocityInterval*5 THEN
					link.yAxisVelocity := TO_DINT((VelocityMmPerSecond + 10 * 2) / 5 * 10000 * 60 );
 
				ELSIF VelocityCounter >= VelocityInterval*5 AND VelocityCounter < VelocityInterval*6 THEN
					link.yAxisVelocity := TO_DINT(-(VelocityMmPerSecond + 10 * 2) / 5 * 10000 * 60);
					
				ELSIF VelocityCounter >= VelocityInterval*6 AND VelocityCounter < VelocityInterval*7 THEN
					link.yAxisVelocity := TO_DINT((VelocityMmPerSecond + 10 * 3) / 5 * 10000 * 60);
					
				ELSIF VelocityCounter >= VelocityInterval*7 AND VelocityCounter < VelocityInterval*8 THEN
					link.yAxisVelocity := TO_DINT(-(VelocityMmPerSecond + 10 * 3) / 5 * 10000 * 60);
					
				ELSIF VelocityCounter >= VelocityInterval*8 AND VelocityCounter < VelocityInterval*9 THEN
					link.yAxisVelocity := TO_DINT((VelocityMmPerSecond + 10 * 4) / 5 * 10000 * 60);
					
				ELSIF VelocityCounter >= VelocityInterval*9 AND VelocityCounter < VelocityInterval*10 THEN
					link.yAxisVelocity := TO_DINT(-(VelocityMmPerSecond + 10 * 4) / 5 * 10000 * 60);
					
				ELSIF VelocityCounter >= VelocityInterval*10 AND VelocityCounter < VelocityInterval*11 THEN
					link.yAxisVelocity := TO_DINT((VelocityMmPerSecond + 10 * 5) / 5 * 10000 * 60);
					
				ELSIF VelocityCounter >= VelocityInterval*11 AND VelocityCounter < VelocityInterval*12 THEN
					link.yAxisVelocity := TO_DINT(-(VelocityMmPerSecond + 10 * 5) / 5 * 10000 * 60);
					
				ELSIF VelocityCounter >= VelocityInterval*12 AND VelocityCounter < VelocityInterval*13 THEN
					link.yAxisVelocity := TO_DINT((VelocityMmPerSecond + 10 * 6) / 5 * 10000 * 60);
					
				ELSIF VelocityCounter >= VelocityInterval*13 AND VelocityCounter < VelocityInterval*14 THEN
					link.yAxisVelocity := TO_DINT(-(VelocityMmPerSecond + 10 * 6) / 5 * 10000 * 60);
					
				ELSIF VelocityCounter >= VelocityInterval*14 AND VelocityCounter < VelocityInterval*15 THEN
					link.yAxisVelocity := TO_DINT((VelocityMmPerSecond + 10 * 7) / 5 * 10000 * 60);
					
				ELSIF VelocityCounter >= VelocityInterval*15 AND VelocityCounter < VelocityInterval*16 THEN
					link.yAxisVelocity := TO_DINT(-(VelocityMmPerSecond + 10 * 7) / 5 * 10000 * 60);
					
				ELSIF VelocityCounter >= VelocityInterval*16 AND VelocityCounter < VelocityInterval*17 THEN
					link.yAxisVelocity := TO_DINT((VelocityMmPerSecond + 10 * 8) / 5 * 10000 * 60);
					
				ELSIF VelocityCounter >= VelocityInterval*17 AND VelocityCounter < VelocityInterval*18 THEN
					link.yAxisVelocity := TO_DINT(-(VelocityMmPerSecond + 10 * 8) / 5 * 10000 * 60);
					
				ELSIF VelocityCounter >= VelocityInterval*18 AND VelocityCounter < VelocityInterval*19 THEN
					link.yAxisVelocity := TO_DINT((VelocityMmPerSecond + 10 * 9) / 5 * 10000 * 60);
					
				ELSIF VelocityCounter >= VelocityInterval*19 AND VelocityCounter < VelocityInterval*20 THEN
					link.yAxisVelocity := TO_DINT(-(VelocityMmPerSecond + 10 * 9) / 5 * 10000 * 60);
					
				ELSIF VelocityCounter >= VelocityInterval*20 AND VelocityCounter < VelocityInterval*21 THEN
					link.yAxisVelocity := TO_DINT((VelocityMmPerSecond + 10 * 10) / 5 * 10000 * 60);
					
				ELSIF VelocityCounter >= VelocityInterval*21 AND VelocityCounter < VelocityInterval*22 THEN
					link.yAxisVelocity := TO_DINT(-(VelocityMmPerSecond + 10 * 10) / 5 * 10000 * 60);
					
				ELSIF VelocityCounter >= VelocityInterval*22 THEN
					link.yAxisVelocity := 0;
					startVelocity := 0;
					state := 60;
					
				END_IF
			ELSE
				state := 60;
			END_IF
			
60 :
	startVelocity:= FALSE;
	state :=0;
	VelocityCounter := 0;
END_CASE

END_PROGRAM

// ---- POUs/ControlParameters.TcPOU
PROGRAM ControlParameters
VAR
END_VAR

END_PROGRAM

// ---- POUs/TorqueCounnter.TcPOU
PROGRAM TorqueCounnter
VAR
	startTest: BOOL:=FALSE;
	i :INT:=1;
	Torque_Nm: INT:=5;
	j: INT:=14;
	TorqueCounter: INT:=0;
	TorqInterval  : INT:=100;
	n: INT;
END_VAR

IF startTest THEN
				TorqueCounter := TorqueCounter + 1;
				
				IF   TorqueCounter >= TorqInterval*(i-1) AND TorqueCounter <TorqInterval*i THEN
					 IF i<=j/2 THEN
						FOR i:=1 TO j/2 BY 1 DO	
							
								IF i MOD 2=1 THEN
								link.torqueX := TO_INT(Torque_Nm * i/2.37*1000);
								ELSE
								link.torqueX := TO_INT(-Torque_Nm * i/2.37*1000);	
	 							END_IF
								
							
						 END_FOR
					   ELSIF i>j/2 THEN
	  					FOR i:=j TO j/2 BY -1 DO	
							IF i MOD 2=1 THEN
								link.torqueX := TO_INT(Torque_Nm * i/2.37*1000);
							ELSE
								link.torqueX := TO_INT(-Torque_Nm * i/2.37*1000);	
	 						END_IF							
						 END_FOR
						
					END_IF					
					
				END_IF				
						
			ELSE
		link.torqueX := 0;
		startTest := FALSE;
		TorqueCounter := 0; 	
END_IF

END_PROGRAM
